{attribute 'linkalways'} 
{attribute 'no_explicit_call' := 'This FB is a CLASS and must be accessed using methods or properties'}
{attribute 'enable_dynamic_creation'}
FUNCTION_BLOCK NodePrototype EXTENDS Disposable IMPLEMENTS I_NodePrototype
VAR
	_path : T_MAXSTRING;
	_node : I_Node;
END_VAR

METHOD PUBLIC Accept
VAR_INPUT
	Visitor : I_NodePrototypeVisitor;
END_VAR
Visitor.VisitNodePrototype(THIS^);
END_METHOD

METHOD PUBLIC Clone : I_Node
VAR_INPUT
END_VAR
Clone := _node.Clone();
END_METHOD

METHOD FB_init : BOOL
VAR_INPUT
	bInitRetains : BOOL; // if TRUE, the retain variables are initialized (warm start / cold start)
	bInCopyCode : BOOL;  // if TRUE, the instance afterwards gets moved into the copy code (online change)
	Path : T_MAXSTRING;
	Node : I_Node;
END_VAR
_path := Path;
_node := Node;
END_METHOD

PROPERTY PUBLIC Node : I_Node
GET
Node := _node;
END_GET
END_PROPERTY

PROPERTY PUBLIC Path : T_MAXSTRING
GET
Path := _path;
END_GET
END_PROPERTY

END_FUNCTION_BLOCK

(* stored: Version 1.1.0.1, ProductVersion 3.1.4024.13
   POU NodePrototype: Id {55dc7f94-c1e6-467e-bf2f-6027928ce074}, SpecialFunc None
   Folder Constructor: Id {58ae38fd-1684-4215-8d1e-e680462ff56d}
   Method Accept: Id {1a99a20e-aedc-429b-befc-14f4054c7a82}
   Method Clone: Id {d1c6cf2a-5559-4198-8f05-596e9b2cccb4}
   Method FB_init: Id {80c1dd88-715a-4de4-ac62-05497ade383c}
   Property Node: Id {94dbaad0-819a-44a5-9024-04676fdd0fee}
   Get Get: Id {c690bf1e-51db-4376-9b60-8b3ee9977859}
   Property Path: Id {c9487224-8d2d-42de-ac8f-a0ebce872a91}
   Get Get: Id {aedc72d9-5311-43eb-abf6-e2311e22985e} *)
